FUNCTION_BLOCK IncrementVarInst
VAR
END_VAR

METHOD Increment : INT
VAR_INST
	nValue	: INT := 5;
END_VAR
nValue := nValue + 1;
Increment := nValue;
END_METHOD

END_FUNCTION_BLOCK

(* stored: Version 1.1.0.1
   POU IncrementVarInst: Id {1d541673-827b-4b8e-b6e0-283c8158f18c}, SpecialFunc None
   Method Increment: Id {3d7c8690-d579-47e3-9748-3bb1390e3174} *)
